(* PLC project OOP_Curso, Beckhoff Automation GmbH TwinCAT PLC Control 3.5.13.21 *)
(* stored: creationDateTime 2023-10-14T20:45:05.5390361, modificationDateTime 2023-10-14T20:45:05.5429384 *)

(* global variable list GVL_1 *)
{attribute 'qualified_only'}
VAR_GLOBAL
	variable1 : BOOL;
	VarInt: INT;
END_VAR

INTERFACE ITF_Profesor
METHOD Fichar
VAR_INPUT
END_VAR
END_METHOD
PROPERTY Salida : int
END_PROPERTY
END_INTERFACE

FUNCTION_BLOCK Persona
VAR_INPUT
END_VAR
VAR_OUTPUT
END_VAR
VAR
END_VAR

            
          

METHOD Comer
VAR_INPUT
END_VAR
                  
                
END_METHOD

PROPERTY DNI : string
GET
VAR
END_VAR
                    
                  
END_GET
SET
VAR
END_VAR
                    
                  
END_SET
END_PROPERTY
END_FUNCTION_BLOCK

FUNCTION_BLOCK Profesor EXTENDS Persona IMPLEMENTS ITF_Profesor
VAR_INPUT
END_VAR
VAR_OUTPUT
END_VAR
VAR
	_Nombre: STRING;
END_VAR

            
          

METHOD DarClases
VAR_INPUT
END_VAR
                  
                
END_METHOD

{warning 'Agregar implementación de método'}
METHOD Fichar
                  
                
END_METHOD

PROPERTY Nombre : String
GET
VAR
END_VAR
                    
                  
END_GET
SET
VAR
END_VAR
                    
                  
END_SET
END_PROPERTY

{warning 'Agregar implementación de propiedad'}
PROPERTY Salida : INT
GET
VAR
END_VAR
                    
                  
END_GET
SET
VAR
END_VAR
                    
                  
END_SET
END_PROPERTY
END_FUNCTION_BLOCK
